FUNCTION_BLOCK FB_ComponentAuto EXTENDS FB_Component
VAR_INPUT
END_VAR
VAR_OUTPUT
END_VAR
VAR
END_VAR

METHOD PROTECTED M_Aborted : BOOL (* Return*)
M_Aborted:= True;
END_METHOD

METHOD PROTECTED M_Execute : BOOL
VAR_INPUT
END_VAR
M_Execute:= True;
END_METHOD

METHOD PROTECTED M_Stopped : BOOL (* Return*)
M_Stopped:= True;
END_METHOD

METHOD PROTECTED N_Holded : BOOL (* Return*)
N_Holded:= True;
END_METHOD

END_FUNCTION_BLOCK

(* stored: Version 1.1.0.1
   POU FB_ComponentAuto: Id {7c7acc8a-6f0b-0aa3-2b16-e85279a26443}, SpecialFunc None
   Method M_Aborted: Id {eeb82b43-bcc8-0c9b-1481-bd5bf2db4bcf}
   Method M_Execute: Id {a6e2a60f-133a-04c9-0c57-a6176e774dfa}
   Method M_Stopped: Id {ba77014d-3704-01e3-2b81-84cca842cbf0}
   Method N_Holded: Id {21fc28f9-c87c-00e7-19fb-5684fb61710c} *)
